ABB RobotStudio station: SC_Conveyor.rspag

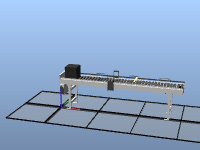
Station conveyor (saved by RobotStudio 7.0.8504.151)
Layout (positions relative to the parent item):
  - 400_guide [part, from Equipment\Conveyor Guide 400.rslib]
  - caja [part] at (125, 0, 780) mm
  - conveyor [smart component]
      signals: DI nueva_caja
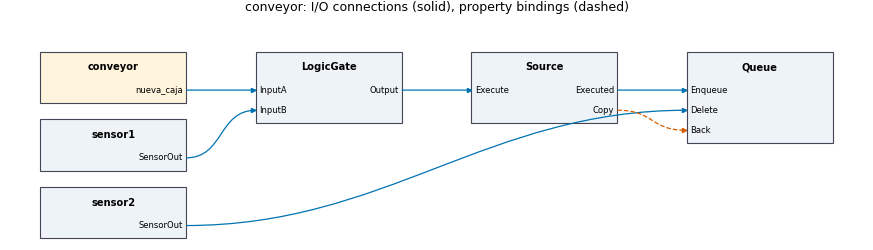
      connections:
        conveyor.nueva_caja -> LogicGate.InputA
        sensor1.SensorOut -> LogicGate.InputB
        LogicGate.Output -> Source.Execute
        Source.Executed -> Queue.Enqueue
        sensor2.SensorOut -> Queue.Delete
        Source.Copy => Queue.Back
    - sensor1 [smart component, from Components\LineSensor.rslib] at (237.02, 0, 871.36) mm
        properties: Start=[0 0 -0.0229730678804657]; End=[0 0.4 -0.0229730678804657]; Radius=0; SensedPart=caja; SensedPoint=[0.237016403198242 0.300000030517578 0.848391052246094]
      - _sensorPart_ [part]
    - sensor2 [smart component, from Components\LineSensor.rslib] at (1862.26, 0, 853.8) mm
        properties: Start=[0 0 0]; End=[0 0.4 0]; Radius=0; SensedPart=(none); SensedPoint=[0 0 0]
      - _sensorPart_ [part]
    - LinearMover [smart component, from Components\LinearMover.rslib]
        properties: Object=Queue; Direction=[1.5 0 0]; Speed=0.3; Reference=Global; ReferenceObject=(none)
    - Queue [smart component, from Components\Queue.rslib]
        properties: Back=(none); Front=(none); Queue={9fa243db-5bcd-4974-8731-7f912ca08678}; NumberOfObjects=0
    - Source [smart component, from Components\Source.rslib]
        properties: Source=caja; Copy=(none); Parent=(none); Position=[0.125 0 0.78]; Orientation=[0 0 0]; Transient=false; PhysicsBehavior=0
    - LogicGate [smart component, from Components\LogicGate.rslib]
        properties: Operator=AND; Delay=0
